PROGRAM MAIN
VAR
	EventBuffer : FB_EventBuffer;
	
	bAddEvent : BOOL;
	stEventToAdd : ST_Event;
	bEventToAddError : BOOL;
	
	
	bReadAndRemoveEvent : BOOL;
	stLastReadEvent : ST_Event;
	bLastEventToReadError : BOOL;
END_VAR

IF bAddEvent THEN
	EventBuffer.AddEvent(stEvent := stEventToAdd, bError => bEventToAddError);
	bAddEvent := FALSE;
END_IF
IF bReadAndRemoveEvent THEN
	EventBuffer.GetAndRemoveEvent(stEvent => stLastReadEvent, bError => bLastEventToReadError);
	bReadAndRemoveEvent := FALSE;
END_IF

END_PROGRAM

(* stored: Version 1.1.0.1, ProductVersion 3.1.4024.12
   POU MAIN: Id {6f43bdf5-072a-481f-8ab2-1f4034213bf6}, SpecialFunc None *)
